FUNCTION_BLOCK FB_Tuning
VAR_INPUT
	bReset: BOOL;
	Axis: AXIS_REF;
	fDeadBand: LREAL;
	fEncRes: LREAL;
END_VAR
VAR_OUTPUT
	nSettleCount: UINT;
	nMaxSettleCount: UINT;
	fMaxFollowerError: LREAL;
	fMaxFollowerErrorCount: LREAL;
END_VAR
VAR
	
END_VAR

IF bReset THEN
	bReset := FALSE;
	nMaxSettleCount := 0;
	fMaxFollowerError := 0;
END_IF

Axis.ReadStatus();
// Settle time calculation
IF Axis.Status.NotMoving THEN
	IF ABS(Axis.NcToPlc.PosDiff) >= fDeadband THEN
		nSettleCount := nSettleCount + 1;
	END_IF
ELSE
	nSettleCount := 0;
END_IF
IF nSettleCount > nMaxSettleCount THEN
	nMaxSettleCount := nSettleCount;
END_IF

IF ABS(Axis.NcToPlc.PosDiff) > fMaxFollowerError THEN
	fMaxFollowerError := ABS(Axis.NcToPlc.PosDiff);
	fMaxFollowerErrorCount := fMaxFollowerError / fEncRes;
END_IF

END_FUNCTION_BLOCK

(* stored: Version 1.1.0.1, ProductVersion 3.1.4020.14
   POU FB_Tuning: Id {60cb0d99-d743-4cf9-88e5-d9f3659b8aa0}, SpecialFunc None *)
